TYPE U_NCI_STATE :
UNION

  stState             : ARRAY[1..MAX_NCI_CH] OF ST_NCI_STATE;

{IF defined (NCI_MAP)}
  {info 'U_NCI_STATE mapping activated'}
  byState   AT %Q*    : ARRAY[1..MAX_NCI_CH] OF
                        ARRAY[1..SIZEOF(ST_NCI_STATE)] OF BYTE;
{ELSE}
  byState             : ARRAY[1..MAX_NCI_CH] OF
                        ARRAY[1..SIZEOF(ST_NCI_STATE)] OF BYTE;
{END_IF}
END_UNION
END_TYPE

(* stored: Version 1.1.0.1, ProductVersion 3.1.4026.13
   DUT U_NCI_STATE: Id {9b8e352c-e3e1-45c0-a459-bd2e18ff0cf6} *)
